		// Module control overrides external ServiceCtrl outside Execute
		AssertTrue(Condition := StoppingModule.PackMLOut.eStateCurrent = E_PackMLState.Stopping, Message := 'Module Stop must enter Stopping.');
		AssertTrue(Condition := StoppingModule.ServiceStatus.SpinAxisMoveAbs.PackMLOut.eStateCurrent = E_PackMLState.Stopping, Message := 'Active MoveAbs Service must enter Stopping.');
		AssertFalse(Condition := SpinAxis.M_IsResourceOwner(OwnerId := E_Chamber1ServiceId.SpinAxisJogCW), Message := 'External Jog Start must be ignored during Module Stopping.');
		AssertTrue(Condition := SpinAxis.M_IsResourceOwner(OwnerId := E_Chamber1ServiceId.SpinAxisMoveAbs), Message := 'MoveAbs must retain ownership while Stop is pending.');
		AssertTrue(Condition := StoppingModule.ModuleStatus.ResponseId = 3001, Message := 'Module must acknowledge the Stop RequestId.');

		// MoveAbs withdrawal must precede physical Stop
		AssertTrue(Condition := StoppingSpinFake.M_GetCall(Index := nHistoryBeforeStopping + 1, CallRecord => MoveWithdrawalCall), Message := 'Module Stop must record MoveAbs withdrawal.');
		AssertTrue(Condition := MoveWithdrawalCall.Operation = E_FakeAxisOperation.MoveAbs, Message := 'Stopping must withdraw MoveAbs before Stop.');
		AssertTrue(Condition := MoveWithdrawalCall.Accepted AND NOT MoveWithdrawalCall.Execute, Message := 'MoveAbs withdrawal must be accepted before ownership release.');
		AssertTrue(Condition := StoppingSpinFake.M_GetCall(Index := nHistoryBeforeStopping + 2, CallRecord => StopCall), Message := 'Module Stop must record physical Stop.');
		AssertTrue(Condition := StopCall.Operation = E_FakeAxisOperation.Stop, Message := 'Physical Stop must follow MoveAbs withdrawal.');
		AssertTrue(Condition := StopCall.Accepted AND StopCall.Execute, Message := 'Physical Stop must be active and accepted.');
		nPhase := 10;

	10:
		// Stop is still pending; script publishes Done after this BaseUnit update
		StoppingModule(
			ModuleCtrl:= ModuleCtrl,
			SystemContext:= SystemContext,
			HeartbeatIndex:= ,
			RuntimeConfig:= RuntimeConfig,
			VariableNodeReader:= VariableNodeReader,
			ServiceCtrl:= ServiceCtrl,
			ServiceParam:= ServiceParam,
			SpinAxis_BaseUnit:= SpinAxis,
			LiftPinAxis_BaseUnit:= LiftAxis);

		AssertTrue(Condition := StoppingModule.PackMLOut.eStateCurrent = E_PackMLState.Stopping, Message := 'Module must wait while a Service Stop is pending.');
		AssertTrue(Condition := StoppingModule.ServiceStatus.SpinAxisMoveAbs.PackMLOut.eStateCurrent = E_PackMLState.Stopping, Message := 'MoveAbs Service must wait for Stop Done.');
		AssertTrue(Condition := SpinAxis.M_IsResourceOwner(OwnerId := E_Chamber1ServiceId.SpinAxisMoveAbs), Message := 'Pending Stop must retain Spin Axis ownership.');
		nPhase := 11;

	11:
		// Service observes Stop Done and performs cleanup
		StoppingModule(
			ModuleCtrl:= ModuleCtrl,
			SystemContext:= SystemContext,
			HeartbeatIndex:= ,
			RuntimeConfig:= RuntimeConfig,
			VariableNodeReader:= VariableNodeReader,
			ServiceCtrl:= ServiceCtrl,
			ServiceParam:= ServiceParam,
			SpinAxis_BaseUnit:= SpinAxis,
			LiftPinAxis_BaseUnit:= LiftAxis);

		// Module waits one additional scan to observe updated ServiceStatus
		AssertTrue(Condition := StoppingModule.PackMLOut.eStateCurrent = E_PackMLState.Stopping, Message := 'Module must remain Stopping until the next scan observes every Service Stopped.');
		AssertTrue(Condition := StoppingModule.ServiceStatus.SpinAxisMoveAbs.PackMLOut.eStateCurrent = E_PackMLState.Stopped, Message := 'Stop Done must move the active Service to Stopped.');
		AssertFalse(Condition := SpinAxis.M_IsResourceOwner(OwnerId := E_Chamber1ServiceId.SpinAxisMoveAbs), Message := 'Stop Done must release Spin Axis ownership.');
		AssertTrue(Condition := StoppingSpinFake.M_GetCall(Index := StoppingSpinFake.HistoryCount, CallRecord => StopCall), Message := 'Stop falling edge must be recorded.');
		AssertTrue(Condition := (StopCall.Operation = E_FakeAxisOperation.Stop) AND StopCall.Accepted AND NOT StopCall.Execute, Message := 'Service must withdraw Stop before releasing ownership.');
		nPhase := 12;

	12:
		// Module observes every Service Stopped
		StoppingModule(
			ModuleCtrl:= ModuleCtrl,
			SystemContext:= SystemContext,
			HeartbeatIndex:= ,
			RuntimeConfig:= RuntimeConfig,
			VariableNodeReader:= VariableNodeReader,
			ServiceCtrl:= ServiceCtrl,
			ServiceParam:= ServiceParam,
			SpinAxis_BaseUnit:= SpinAxis,
			LiftPinAxis_BaseUnit:= LiftAxis);

		AssertTrue(Condition := StoppingModule.PackMLOut.eStateCurrent = E_PackMLState.Stopped, Message := 'Module must reach Stopped only after every Service is Stopped.');
		AssertTrue(
			Condition := (StoppingModule.ServiceStatus.SpinAxisJogCW.PackMLOut.eStateCurrent = E_PackMLState.Stopped)
				AND (StoppingModule.ServiceStatus.SpinAxisMoveAbs.PackMLOut.eStateCurrent = E_PackMLState.Stopped)
				AND (StoppingModule.ServiceStatus.SpinAxisMoveVelCW.PackMLOut.eStateCurrent = E_PackMLState.Stopped)
				AND (StoppingModule.ServiceStatus.LiftPinAxisMoveVelCW.PackMLOut.eStateCurrent = E_PackMLState.Stopped)
				AND (StoppingModule.ServiceStatus.LiftPinAxisMoveVelCCW.PackMLOut.eStateCurrent = E_PackMLState.Stopped)
				AND (StoppingModule.ServiceStatus.LiftPinAxisMoveAbs.PackMLOut.eStateCurrent = E_PackMLState.Stopped),
			Message := 'Module Stopped requires every Service Stopped.');
		AssertFalse(Condition := SpinAxis.M_IsResourceOwner(OwnerId := E_Chamber1ServiceId.SpinAxisMoveAbs), Message := 'Stopped Module must not retain Spin Axis ownership.');
		AssertFalse(Condition := SpinAxis.M_IsResourceOwner(OwnerId := E_Chamber1ServiceId.SpinAxisJogCW), Message := 'Ignored external Jog Start must not acquire ownership later.');
		nPhase := 0;

		TEST_FINISHED();
END_CASE
END_METHOD

END_FUNCTION_BLOCK

// ---- POUs/10_Chamber1/FB_Chamber1_Module.TcPOU
FUNCTION_BLOCK FB_Chamber1_Module EXTENDS FB_ModuleBase
VAR_INPUT	
	HwInput : ST_Chamber1_Signal_In;

	ServiceCtrl : REFERENCE TO ST_Chamber1_ServiceCtrl;
	ServiceParam : REFERENCE TO ST_Chamber1_ServiceParam;

	// Base unit used in Chamber1 chamber
	SpinAxis_BaseUnit : I_Axis_BaseUnit;
	LiftPinAxis_BaseUnit : I_Axis_BaseUnit;
END_VAR

VAR_OUTPUT
	HwOutput : ST_Chamber1_Signal_Out;
	ServiceStatus : ST_Chamber1_ServiceStatus;
END_VAR

VAR
	_EffectiveServiceCtrl : ST_Chamber1_ServiceCtrl;
	_EffectiveServiceParam : ST_Chamber1_ServiceParam;
	_ServiceStatusStore : ST_Chamber1_ServiceStatus;

	_SpinAxisJogCWService : FB_Chamber1SpinAxisJogCWServices;
	_SpinAxisMoveAbsService : FB_Chamber1SpinAxisMoveAbsServices;
	_SpinAxisMoveVelCWService : FB_Chamber1SpinAxisMoveVelCWServices;
	_LiftPinAxisMoveVelCWService : FB_Chamber1LiftPinAxisMoveVelCWServices;
	_LiftPinAxisMoveVelCCWService : FB_Chamber1LiftPinAxisMoveVelCCWServices;
	_LiftPinAxisMoveAbsService : FB_Chamber1LiftPinAxisMoveAbsServices;
	_WaferSendService : FB_Chamber1WaferSendService;
	_WaferReceiveService : FB_Chamber1WaferReceiveService;
	_PreparePositionService : FB_Chamber1PreparePositionService;

END_VAR

// An unbound Axis interface is a composition error. Keep the Module inert.
IF (SpinAxis_BaseUnit = 0) OR (LiftPinAxis_BaseUnit = 0) THEN
	RETURN;
END_IF

// Config wafer transfer endpoint
ModuleStatus.WaferTransferResponseList[1].EndpointId := 1;
ModuleStatus.WaferTransferResponseList[1].WaferHandlingType := E_WaferHandlingType.Passive;
ModuleStatus.WaferTransferResponseList[1].Capability := E_TransferCapability.Bidirectional;
ModuleStatus.WaferTransferResponseList[1].SendServiceId := E_Chamber1ServiceId.WaferSend;
ModuleStatus.WaferTransferResponseList[1].ReceiveServiceId := E_Chamber1ServiceId.WaferReceive;

M_UpdateModule();

// Update status
ServiceStatus := _ServiceStatusStore;

// Link status to module
ModuleStatus.WaferTransferResponseList[1].Send.Status := ServiceStatus.WaferSend;
ModuleStatus.WaferTransferResponseList[1].Send.Signal := _WaferSendService.SignalOut;
ModuleStatus.WaferTransferResponseList[1].SendReady := _ServiceCoordinator.AllIdle;
ModuleStatus.WaferTransferResponseList[1].Receive.Status := ServiceStatus.WaferReceive;
ModuleStatus.WaferTransferResponseList[1].Receive.Signal := _WaferReceiveService.SignalOut;
ModuleStatus.WaferTransferResponseList[1].ReceiveReady := _ServiceCoordinator.AllIdle;

METHOD PROTECTED H_RegisterServices
// Register services
M_RegisterService(
	ServiceId := E_Chamber1ServiceId.SpinAxisJogCW,
	AllowCompositeCall := TRUE,
	UpperCtrl := ServiceCtrl.SpinAxisJogCW,
	EffectiveCtrl := _EffectiveServiceCtrl.SpinAxisJogCW,
	UpperParam := ServiceParam.SpinAxisJogCW,
	EffectiveParam := _EffectiveServiceParam.SpinAxisJogCW,
	Status := _ServiceStatusStore.SpinAxisJogCW);
M_RegisterService(
	ServiceId := E_Chamber1ServiceId.SpinAxisMoveAbs,
	AllowCompositeCall := TRUE,
	UpperCtrl := ServiceCtrl.SpinAxisMoveAbs,
	EffectiveCtrl := _EffectiveServiceCtrl.SpinAxisMoveAbs,
	UpperParam := ServiceParam.SpinAxisMoveAbs,
	EffectiveParam := _EffectiveServiceParam.SpinAxisMoveAbs,
	Status := _ServiceStatusStore.SpinAxisMoveAbs);
M_RegisterService(
	ServiceId := E_Chamber1ServiceId.SpinAxisMoveVelCW,
	AllowCompositeCall := TRUE,
	UpperCtrl := ServiceCtrl.SpinAxisMoveVelCW,
	EffectiveCtrl := _EffectiveServiceCtrl.SpinAxisMoveVelCW,
	UpperParam := ServiceParam.SpinAxisMoveVelCW,
	EffectiveParam := _EffectiveServiceParam.SpinAxisMoveVelCW,
	Status := _ServiceStatusStore.SpinAxisMoveVelCW);
M_RegisterService(
	ServiceId := E_Chamber1ServiceId.LiftPinAxisMoveVelCW,
	AllowCompositeCall := TRUE,
	UpperCtrl := ServiceCtrl.LiftPinAxisMoveVelCW,
	EffectiveCtrl := _EffectiveServiceCtrl.LiftPinAxisMoveVelCW,
	UpperParam := ServiceParam.LiftPinAxisMoveVelCW,
	EffectiveParam := _EffectiveServiceParam.LiftPinAxisMoveVelCW,
	Status := _ServiceStatusStore.LiftPinAxisMoveVelCW);
M_RegisterService(
	ServiceId := E_Chamber1ServiceId.LiftPinAxisMoveVelCCW,
	AllowCompositeCall := TRUE,
	UpperCtrl := ServiceCtrl.LiftPinAxisMoveVelCCW,
	EffectiveCtrl := _EffectiveServiceCtrl.LiftPinAxisMoveVelCCW,
	UpperParam := ServiceParam.LiftPinAxisMoveVelCCW,
	EffectiveParam := _EffectiveServiceParam.LiftPinAxisMoveVelCCW,
	Status := _ServiceStatusStore.LiftPinAxisMoveVelCCW);
M_RegisterService(
	ServiceId := E_Chamber1ServiceId.LiftPinAxisMoveAbs,
	AllowCompositeCall := TRUE,
	UpperCtrl := ServiceCtrl.LiftPinAxisMoveAbs,
	EffectiveCtrl := _EffectiveServiceCtrl.LiftPinAxisMoveAbs,
	UpperParam := ServiceParam.LiftPinAxisMoveAbs,
	EffectiveParam := _EffectiveServiceParam.LiftPinAxisMoveAbs,
	Status := _ServiceStatusStore.LiftPinAxisMoveAbs);
M_RegisterService(
	ServiceId := E_Chamber1ServiceId.WaferSend,
	AllowCompositeCall := FALSE,
	UpperCtrl := ServiceCtrl.WaferSend,
	EffectiveCtrl := _EffectiveServiceCtrl.WaferSend,
	UpperParam := ServiceParam.WaferSend,
	EffectiveParam := _EffectiveServiceParam.WaferSend,
	Status := _ServiceStatusStore.WaferSend);
M_RegisterService(
	ServiceId := E_Chamber1ServiceId.WaferReceive,
	AllowCompositeCall := FALSE,
	UpperCtrl := ServiceCtrl.WaferReceive,
	EffectiveCtrl := _EffectiveServiceCtrl.WaferReceive,
	UpperParam := ServiceParam.WaferReceive,
	EffectiveParam := _EffectiveServiceParam.WaferReceive,
	Status := _ServiceStatusStore.WaferReceive);
M_RegisterService(
	ServiceId := E_Chamber1ServiceId.PreparePosition,
	AllowCompositeCall := FALSE,
	UpperCtrl := ServiceCtrl.PreparePosition,
	EffectiveCtrl := _EffectiveServiceCtrl.PreparePosition,
	UpperParam := ServiceParam.PreparePosition,
	EffectiveParam := _EffectiveServiceParam.PreparePosition,
	Status := _ServiceStatusStore.PreparePosition);

// Register dependency of composite service
_PreparePositionService.M_RegisterDefinition(
	CompositeServiceId := E_Chamber1ServiceId.PreparePosition,
	Coordinator := _ServiceCoordinator);
END_METHOD

METHOD PROTECTED H_UpdateBaseUnit
VAR_INPUT
END_VAR
SpinAxis_BaseUnit.M_CyclicUpdate();
LiftPinAxis_BaseUnit.M_CyclicUpdate();
END_METHOD

METHOD PROTECTED H_UpdateService
VAR_INPUT
END_VAR
_SpinAxisJogCWService(
	Ctrl:= _EffectiveServiceCtrl.SpinAxisJogCW,
	Param:= _EffectiveServiceParam.SpinAxisJogCW,
	Context:= _ServiceContext,
	Axis_BaseUnit:= SpinAxis_BaseUnit,
	// Owner IDs are assigned by the Module so each Service instance is unique.
	ServiceId:= E_Chamber1ServiceId.SpinAxisJogCW,
	Status=> _ServiceStatusStore.SpinAxisJogCW);

_SpinAxisMoveAbsService(
	Ctrl:= _EffectiveServiceCtrl.SpinAxisMoveAbs,
	Param:= _EffectiveServiceParam.SpinAxisMoveAbs,
	Context:= _ServiceContext,
	Axis_BaseUnit:= SpinAxis_BaseUnit,
	ServiceId:= E_Chamber1ServiceId.SpinAxisMoveAbs,
	Status=> _ServiceStatusStore.SpinAxisMoveAbs);

_SpinAxisMoveVelCWService(
	Ctrl:= _EffectiveServiceCtrl.SpinAxisMoveVelCW,
	Param:= _EffectiveServiceParam.SpinAxisMoveVelCW,
	Context:= _ServiceContext,
	Axis_BaseUnit:= SpinAxis_BaseUnit,
	ServiceId:= E_Chamber1ServiceId.SpinAxisMoveVelCW,
	Status=> _ServiceStatusStore.SpinAxisMoveVelCW);

_LiftPinAxisMoveVelCWService(
	Ctrl:= _EffectiveServiceCtrl.LiftPinAxisMoveVelCW,
	Param:= _EffectiveServiceParam.LiftPinAxisMoveVelCW,
	Context:= _ServiceContext,
	Axis_BaseUnit:= LiftPinAxis_BaseUnit,
	ServiceId:= E_Chamber1ServiceId.LiftPinAxisMoveVelCW,
	Status=> _ServiceStatusStore.LiftPinAxisMoveVelCW);

_LiftPinAxisMoveVelCCWService(
	Ctrl:= _EffectiveServiceCtrl.LiftPinAxisMoveVelCCW,
	Param:= _EffectiveServiceParam.LiftPinAxisMoveVelCCW,
	Context:= _ServiceContext,
	Axis_BaseUnit:= LiftPinAxis_BaseUnit,
	ServiceId:= E_Chamber1ServiceId.LiftPinAxisMoveVelCCW,
	Status=> _ServiceStatusStore.LiftPinAxisMoveVelCCW);

_LiftPinAxisMoveAbsService(
	Ctrl:= _EffectiveServiceCtrl.LiftPinAxisMoveAbs,
	Param:= _EffectiveServiceParam.LiftPinAxisMoveAbs,
	Context:= _ServiceContext,
	Axis_BaseUnit:= LiftPinAxis_BaseUnit,
	ServiceId:= E_Chamber1ServiceId.LiftPinAxisMoveAbs,
	Status=> _ServiceStatusStore.LiftPinAxisMoveAbs);

_PreparePositionService(
	Ctrl := _EffectiveServiceCtrl.PreparePosition,
	Param := _EffectiveServiceParam.PreparePosition,
	Context := _ServiceContext,
	ServiceId := E_Chamber1ServiceId.PreparePosition,
	Status => _ServiceStatusStore.PreparePosition);

// Both directions share Station material and hardware storage.
// TODO: Coordinate Send/Receive access when implementing the transfer sequences.
_WaferSendService(
	Ctrl := _EffectiveServiceCtrl.WaferSend,
	Param := _EffectiveServiceParam.WaferSend,
	Context := _ServiceContext,
	ServiceId := E_Chamber1ServiceId.WaferSend,
	MaterialInfo := ModuleStatus.WaferTransferResponseList[1].MaterialInfo,
	SpinAxis_BaseUnit := SpinAxis_BaseUnit,
	LiftPinAxis_BaseUnit := LiftPinAxis_BaseUnit,
	Status => _ServiceStatusStore.WaferSend);

_WaferReceiveService(
	Ctrl := _EffectiveServiceCtrl.WaferReceive,
	Param := _EffectiveServiceParam.WaferReceive,
	Context := _ServiceContext,
	ServiceId := E_Chamber1ServiceId.WaferReceive,
	MaterialInfo := ModuleStatus.WaferTransferResponseList[1].MaterialInfo,
	SpinAxis_BaseUnit := SpinAxis_BaseUnit,
	LiftPinAxis_BaseUnit := LiftPinAxis_BaseUnit,
	Status => _ServiceStatusStore.WaferReceive);
END_METHOD

END_FUNCTION_BLOCK

// ---- POUs/10_Chamber1/Services/FB_Chamber1WaferSendService.TcPOU
FUNCTION_BLOCK FB_Chamber1WaferSendService EXTENDS FB_ServiceBase
VAR_INPUT
	Param : ST_WaferTransferParam;
	SpinAxis_BaseUnit : I_Axis_BaseUnit;
	LiftPinAxis_BaseUnit : I_Axis_BaseUnit;
END_VAR

VAR_IN_OUT
	// Shared with the opposite direction; arbitration belongs to the future transfer flow.
	MaterialInfo : ST_MaterialInfo;
END_VAR

VAR_OUTPUT
	SignalOut : ST_TransferHandshakeSignal;
END_VAR

M_UpdateService(CompletionBehavior := E_ServiceCompletionBehavior.SendWafer);

METHOD PROTECTED H_OnAborting : E_PackMLHookResult
VAR_INPUT
	bFirstScan : BOOL;
END_VAR
// TODO: Implement abort cleanup and material reconciliation for an interrupted transfer.
// The skeleton acquires no resources and issues no hardware commands.
H_OnAborting := E_PackMLHookResult.Done;
END_METHOD

METHOD PROTECTED H_OnCompleting : E_PackMLHookResult
VAR_INPUT
	bFirstScan : BOOL;
END_VAR
// TODO: Finish handshake cleanup and release resources after confirmed completion.
H_OnCompleting := E_PackMLHookResult.Done;
END_METHOD

METHOD PROTECTED H_OnExecute : E_PackMLHookResult
VAR_INPUT
	bFirstScan : BOOL;
END_VAR
// TODO: Implement sending from Chamber1, handshake sequencing, and timeout handling.
// TransferReady advertises Endpoint availability; SignalOut.Ready is a handshake signal.
// TODO: Clear MaterialInfo only after confirmed send completion.
// Keep the skeleton active until Stop/Abort; do not report a completed transfer.
H_OnExecute := E_PackMLHookResult.Busy;
END_METHOD

METHOD PROTECTED H_OnResetting : E_PackMLHookResult
VAR_INPUT
	bFirstScan : BOOL;
END_VAR
MEMSET(ADR(Status.ErrorList), 0, SIZEOF(Status.ErrorList));
// TODO: Reset transfer-local state without unconditionally clearing the Station material.
H_OnResetting := E_PackMLHookResult.Done;
END_METHOD

METHOD PROTECTED H_OnStarting : E_PackMLHookResult
VAR_INPUT
	bFirstScan : BOOL;
END_VAR
// TODO: Validate Param against StationId, latch transfer data, and reserve resources.
H_OnStarting := E_PackMLHookResult.Done;
END_METHOD

METHOD PROTECTED H_OnStopping : E_PackMLHookResult
VAR_INPUT
	bFirstScan : BOOL;
END_VAR
// TODO: Withdraw handshake/motion requests and complete owned-resource cleanup.
// The skeleton acquires no resources and issues no hardware commands.
H_OnStopping := E_PackMLHookResult.Done;
END_METHOD

END_FUNCTION_BLOCK
